(* PLC project  *)

CONFIGURATION EtherCAT_Master_SoftMotion
END_CONFIGURATION
